// Mitsubishi GX Works2 project: RL8_12-03-62 - LossCode   PLC: Q01U

PROGRAM MAIN  // À¯ÁÊßÈÙ
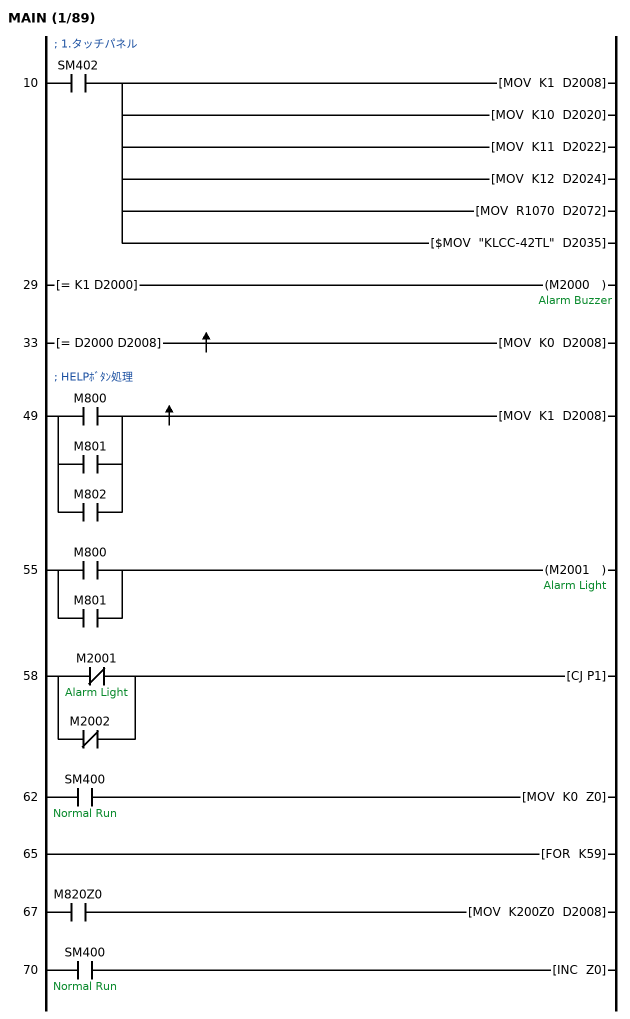
; 1.タッチパネル
; 
10    LD      SM402
      MOV     K1 D2008
      MOV     K10 D2020
      MOV     K11 D2022
      MOV     K12 D2024
      MOV     R1070 D2072
      $MOV    "KLCC-42TL" D2035
29    LD=     K1 D2000
      OUT     M2000  ; Alarm Buzzer
33    LD=     D2000 D2008
      MEP
      MOV     K0 D2008
; HELPﾎﾞﾀﾝ処理
49    LD      M800
      OR      M801
      OR      M802
      MEP
      MOV     K1 D2008
55    LD      M800
      OR      M801
      OUT     M2001  ; Alarm Light
58    LDI     M2001  ; Alarm Light
      ORI     M2002
      CJ      P1
62    LD      SM400  ; Normal Run
      MOV     K0 Z0
65    FOR     K59
67    LD      M820Z0
      MOV     K200Z0 D2008
70    LD      SM400  ; Normal Run
      INC     Z0
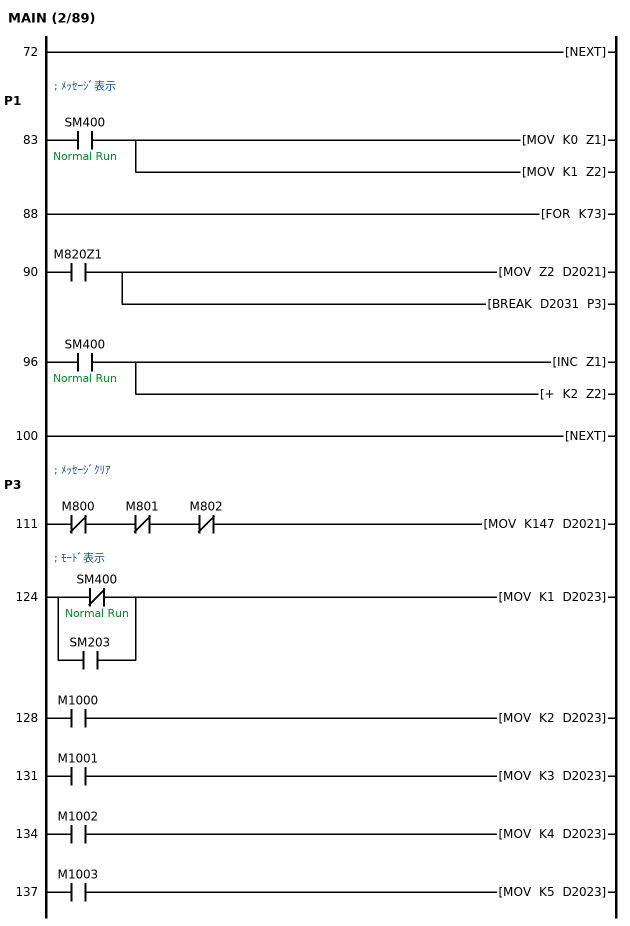
72    NEXT
      P1
; ﾒｯｾｰｼﾞ表示
83    LD      SM400  ; Normal Run
      MOV     K0 Z1
      MOV     K1 Z2
88    FOR     K73
90    LD      M820Z1
      MOV     Z2 D2021
      BREAK   D2031 P3
96    LD      SM400  ; Normal Run
      INC     Z1
      +       K2 Z2
100   NEXT
; ﾒｯｾｰｼﾞｸﾘｱ
      P3
111   LDI     M800
      ANI     M801
      ANI     M802
      MOV     K147 D2021
; ﾓｰﾄﾞ表示
124   LDI     SM400  ; Normal Run
      OR      SM203
      MOV     K1 D2023
128   LD      M1000
      MOV     K2 D2023
131   LD      M1001
      MOV     K3 D2023
134   LD      M1002
      MOV     K4 D2023
137   LD      M1003
      MOV     K5 D2023
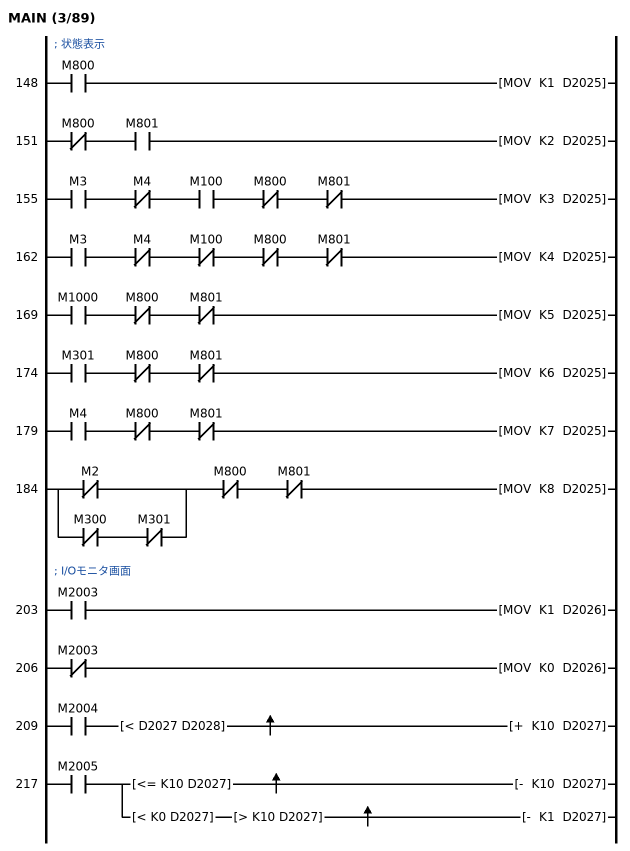
; 状態表示
148   LD      M800
      MOV     K1 D2025
151   LDI     M800
      AND     M801
      MOV     K2 D2025
155   LD      M3
      ANI     M4
      AND     M100
      ANI     M800
      ANI     M801
      MOV     K3 D2025
162   LD      M3
      ANI     M4
      ANI     M100
      ANI     M800
      ANI     M801
      MOV     K4 D2025
169   LD      M1000
      ANI     M800
      ANI     M801
      MOV     K5 D2025
174   LD      M301
      ANI     M800
      ANI     M801
      MOV     K6 D2025
179   LD      M4
      ANI     M800
      ANI     M801
      MOV     K7 D2025
184   LDI     M2
      LDI     M300
      ANI     M301
      ORB
      ANI     M800
      ANI     M801
      MOV     K8 D2025
; I/Oモニタ画面
203   LD      M2003
      MOV     K1 D2026
206   LDI     M2003
      MOV     K0 D2026
209   LD      M2004
      AND<    D2027 D2028
      MEP
      +       K10 D2027
217   LD      M2005
      MPS
      AND<=   K10 D2027
      MEP
      -       K10 D2027
      MPP
      AND<    K0 D2027
      AND>    K10 D2027
      MEP
      -       K1 D2027
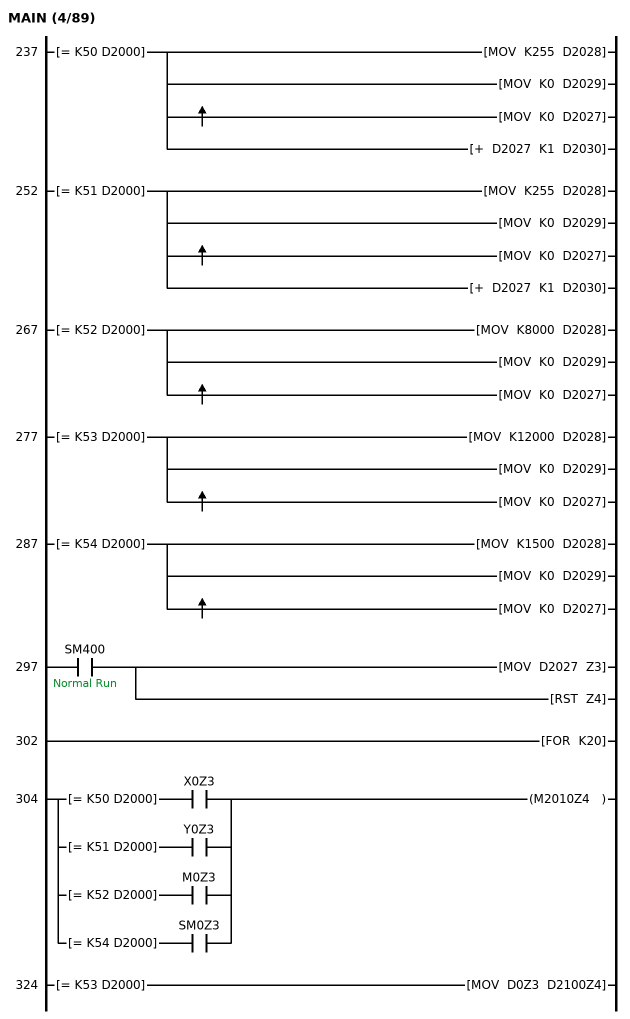
237   LD=     K50 D2000
      MOV     K255 D2028
      MOV     K0 D2029
      MPS
      MEP
      MOV     K0 D2027
      MPP
      +       D2027 K1 D2030
252   LD=     K51 D2000
      MOV     K255 D2028
      MOV     K0 D2029
      MPS
      MEP
      MOV     K0 D2027
      MPP
      +       D2027 K1 D2030
267   LD=     K52 D2000
      MOV     K8000 D2028
      MOV     K0 D2029
      MEP
      MOV     K0 D2027
277   LD=     K53 D2000
      MOV     K12000 D2028
      MOV     K0 D2029
      MEP
      MOV     K0 D2027
287   LD=     K54 D2000
      MOV     K1500 D2028
      MOV     K0 D2029
      MEP
      MOV     K0 D2027
297   LD      SM400  ; Normal Run
      MOV     D2027 Z3
      RST     Z4
302   FOR     K20
304   LD=     K50 D2000
      AND     X0Z3
      LD=     K51 D2000
      AND     Y0Z3
      ORB
      LD=     K52 D2000
      AND     M0Z3
      ORB
      LD=     K54 D2000
      AND     SM0Z3
      ORB
      OUT     M2010Z4
324   LD=     K53 D2000
      MOV     D0Z3 D2100Z4
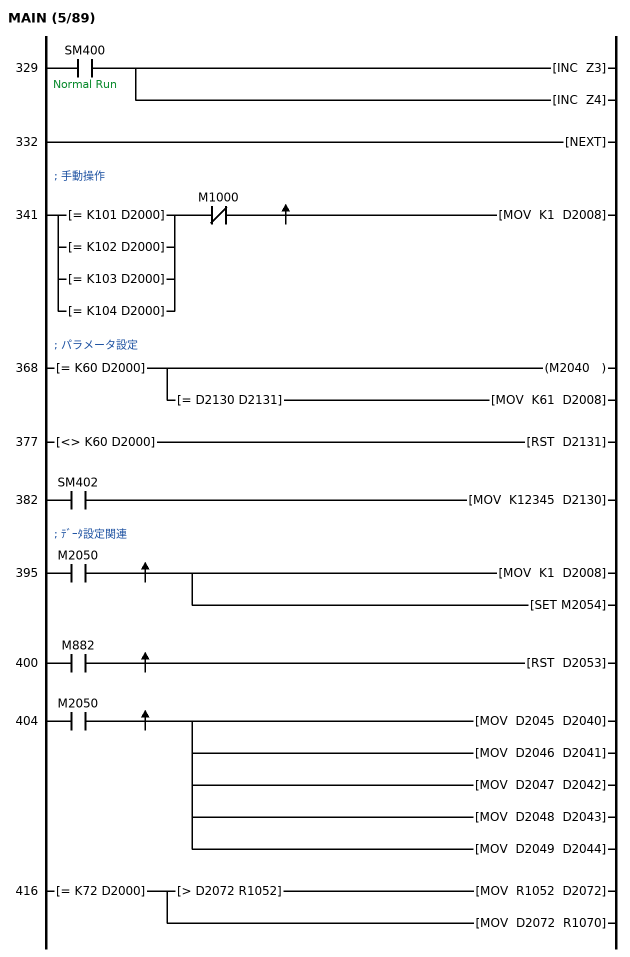
329   LD      SM400  ; Normal Run
      INC     Z3
      INC     Z4
332   NEXT
; 手動操作
341   LD=     K101 D2000
      OR=     K102 D2000
      OR=     K103 D2000
      OR=     K104 D2000
      ANI     M1000
      MEP
      MOV     K1 D2008
; パラメータ設定
368   LD=     K60 D2000
      OUT     M2040
      AND=    D2130 D2131
      MOV     K61 D2008
377   LD<>    K60 D2000
      RST     D2131
382   LD      SM402
      MOV     K12345 D2130
; ﾃﾞｰﾀ設定関連
395   LD      M2050
      MEP
      MOV     K1 D2008
      SET     M2054
400   LD      M882
      MEP
      RST     D2053
404   LD      M2050
      MEP
      MOV     D2045 D2040
      MOV     D2046 D2041
      MOV     D2047 D2042
      MOV     D2048 D2043
      MOV     D2049 D2044
416   LD=     K72 D2000
      MPS
      AND>    D2072 R1052
      MOV     R1052 D2072
      MPP
      MOV     D2072 R1070
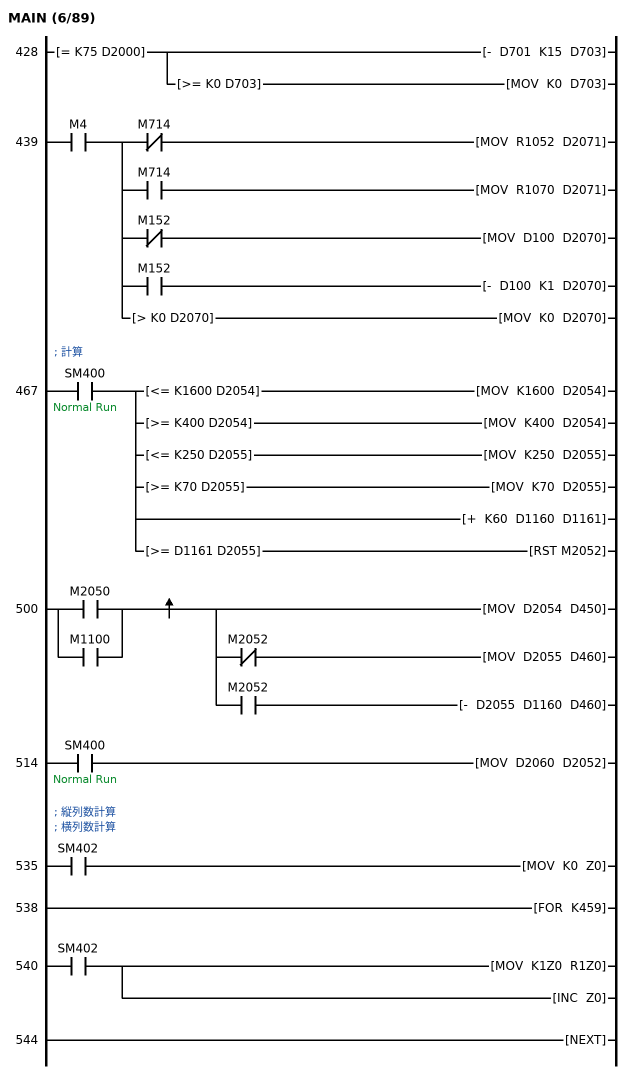
428   LD=     K75 D2000
      -       D701 K15 D703
      AND>=   K0 D703
      MOV     K0 D703
439   LD      M4
      MPS
      ANI     M714
      MOV     R1052 D2071
      MRD
      AND     M714
      MOV     R1070 D2071
      MRD
      ANI     M152
      MOV     D100 D2070
      MRD
      AND     M152
      -       D100 K1 D2070
      MPP
      AND>    K0 D2070
      MOV     K0 D2070
; 計算
467   LD      SM400  ; Normal Run
      MPS
      AND<=   K1600 D2054
      MOV     K1600 D2054
      MRD
      AND>=   K400 D2054
      MOV     K400 D2054
      MRD
      AND<=   K250 D2055
      MOV     K250 D2055
      MRD
      AND>=   K70 D2055
      MOV     K70 D2055
      MPP
      +       K60 D1160 D1161
      AND>=   D1161 D2055
      RST     M2052
500   LD      M2050
      OR      M1100
      MEP
      MOV     D2054 D450
      MPS
      ANI     M2052
      MOV     D2055 D460
      MPP
      AND     M2052
      -       D2055 D1160 D460
514   LD      SM400  ; Normal Run
      MOV     D2060 D2052
; 縦列数計算
; 横列数計算
535   LD      SM402
      MOV     K0 Z0
538   FOR     K459
540   LD      SM402
      MOV     K1Z0 R1Z0
      INC     Z0
544   NEXT
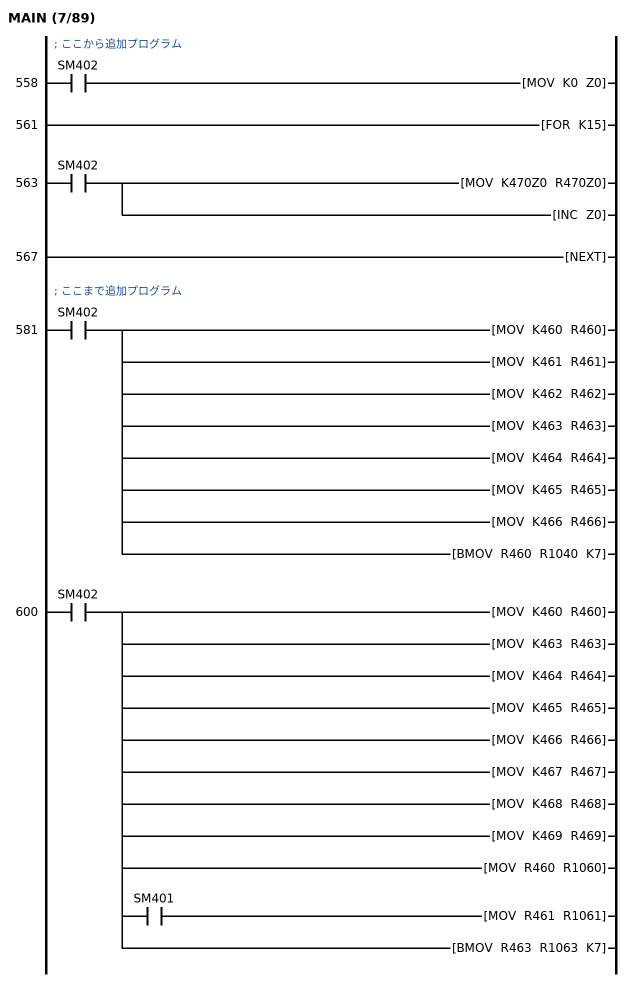
; ここから追加プログラム
558   LD      SM402
      MOV     K0 Z0
561   FOR     K15
563   LD      SM402
      MOV     K470Z0 R470Z0
      INC     Z0
567   NEXT
; ここまで追加プログラム
581   LD      SM402
      MOV     K460 R460
      MOV     K461 R461
      MOV     K462 R462
      MOV     K463 R463
      MOV     K464 R464
      MOV     K465 R465
      MOV     K466 R466
      BMOV    R460 R1040 K7
600   LD      SM402
      MOV     K460 R460
      MOV     K463 R463
      MOV     K464 R464
      MOV     K465 R465
      MOV     K466 R466
      MOV     K467 R467
      MOV     K468 R468
      MOV     K469 R469
      MOV     R460 R1060
      MPS
      AND     SM401
      MOV     R461 R1061
      MPP
      BMOV    R463 R1063 K7
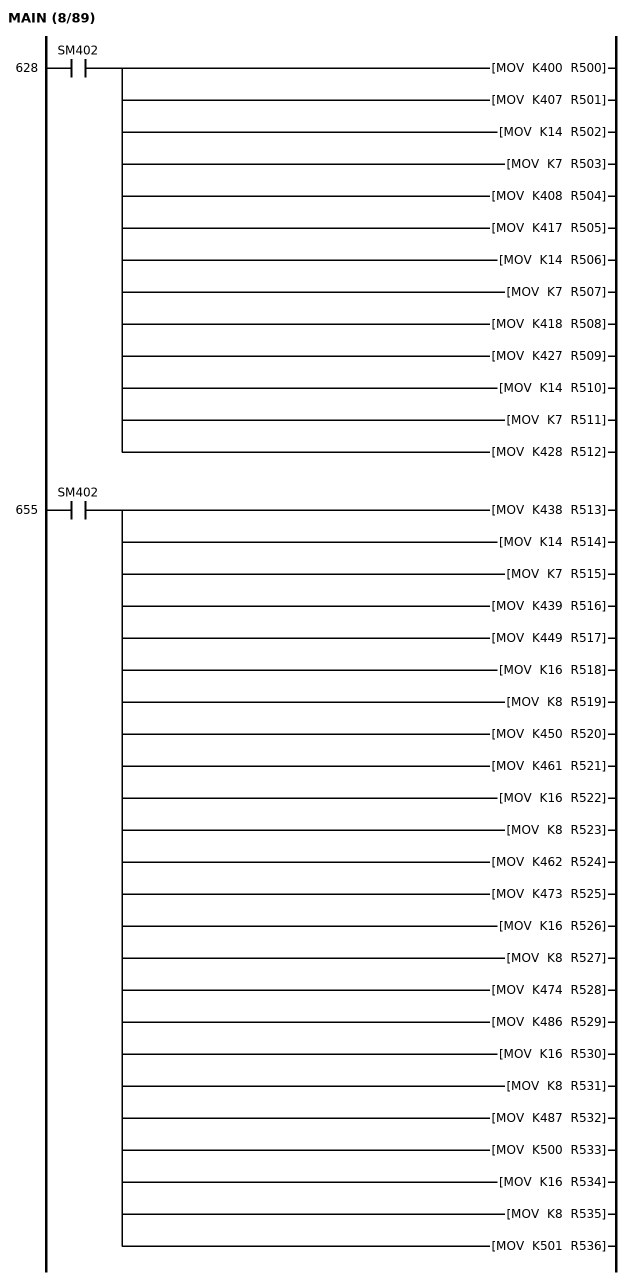
628   LD      SM402
      MOV     K400 R500
      MOV     K407 R501
      MOV     K14 R502
      MOV     K7 R503
      MOV     K408 R504
      MOV     K417 R505
      MOV     K14 R506
      MOV     K7 R507
      MOV     K418 R508
      MOV     K427 R509
      MOV     K14 R510
      MOV     K7 R511
      MOV     K428 R512
655   LD      SM402
      MOV     K438 R513
      MOV     K14 R514
      MOV     K7 R515
      MOV     K439 R516
      MOV     K449 R517
      MOV     K16 R518
      MOV     K8 R519
      MOV     K450 R520
      MOV     K461 R521
      MOV     K16 R522
      MOV     K8 R523
      MOV     K462 R524
      MOV     K473 R525
      MOV     K16 R526
      MOV     K8 R527
      MOV     K474 R528
      MOV     K486 R529
      MOV     K16 R530
      MOV     K8 R531
      MOV     K487 R532
      MOV     K500 R533
      MOV     K16 R534
      MOV     K8 R535
      MOV     K501 R536
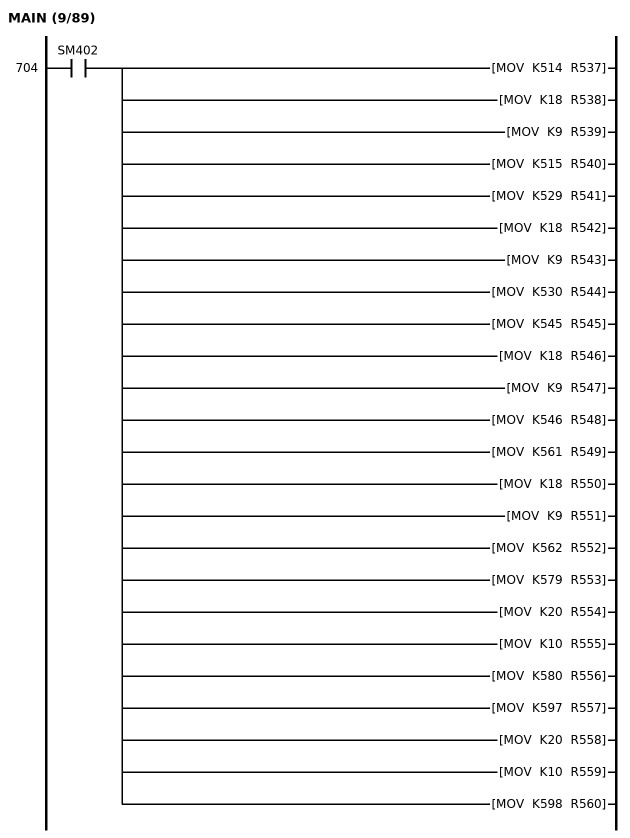
704   LD      SM402
      MOV     K514 R537
      MOV     K18 R538
      MOV     K9 R539
      MOV     K515 R540
      MOV     K529 R541
      MOV     K18 R542
      MOV     K9 R543
      MOV     K530 R544
      MOV     K545 R545
      MOV     K18 R546
      MOV     K9 R547
      MOV     K546 R548
      MOV     K561 R549
      MOV     K18 R550
      MOV     K9 R551
      MOV     K562 R552
      MOV     K579 R553
      MOV     K20 R554
      MOV     K10 R555
      MOV     K580 R556
      MOV     K597 R557
      MOV     K20 R558
      MOV     K10 R559
      MOV     K598 R560
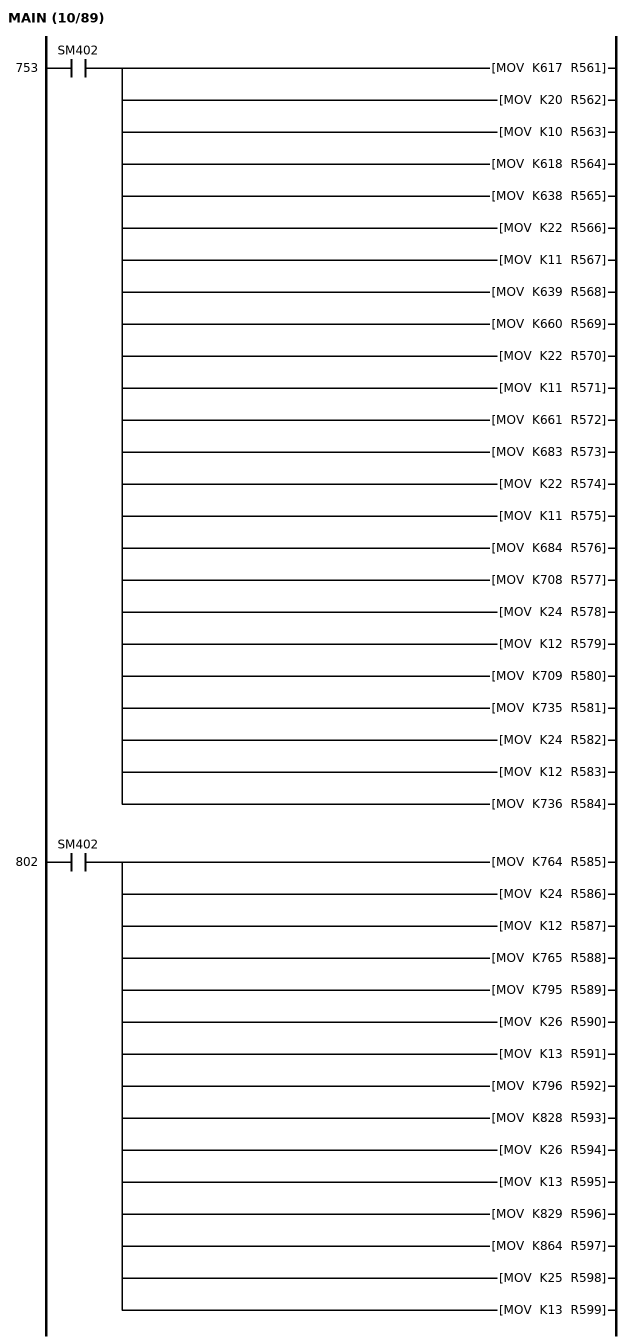
753   LD      SM402
      MOV     K617 R561
      MOV     K20 R562
      MOV     K10 R563
      MOV     K618 R564
      MOV     K638 R565
      MOV     K22 R566
      MOV     K11 R567
      MOV     K639 R568
      MOV     K660 R569
      MOV     K22 R570
      MOV     K11 R571
      MOV     K661 R572
      MOV     K683 R573
      MOV     K22 R574
      MOV     K11 R575
      MOV     K684 R576
      MOV     K708 R577
      MOV     K24 R578
      MOV     K12 R579
      MOV     K709 R580
      MOV     K735 R581
      MOV     K24 R582
      MOV     K12 R583
      MOV     K736 R584
802   LD      SM402
      MOV     K764 R585
      MOV     K24 R586
      MOV     K12 R587
      MOV     K765 R588
      MOV     K795 R589
      MOV     K26 R590
      MOV     K13 R591
      MOV     K796 R592
      MOV     K828 R593
      MOV     K26 R594
      MOV     K13 R595
      MOV     K829 R596
      MOV     K864 R597
      MOV     K25 R598
      MOV     K13 R599
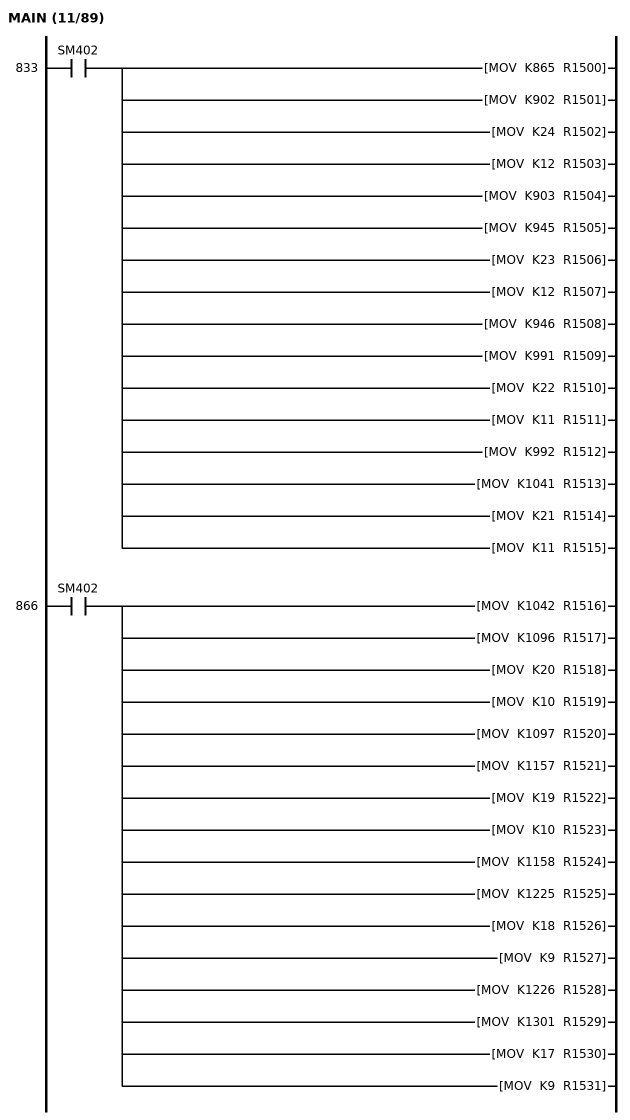
833   LD      SM402
      MOV     K865 R1500
      MOV     K902 R1501
      MOV     K24 R1502
      MOV     K12 R1503
      MOV     K903 R1504
      MOV     K945 R1505
      MOV     K23 R1506
      MOV     K12 R1507
      MOV     K946 R1508
      MOV     K991 R1509
      MOV     K22 R1510
      MOV     K11 R1511
      MOV     K992 R1512
      MOV     K1041 R1513
      MOV     K21 R1514
      MOV     K11 R1515
866   LD      SM402
      MOV     K1042 R1516
      MOV     K1096 R1517
      MOV     K20 R1518
      MOV     K10 R1519
      MOV     K1097 R1520
      MOV     K1157 R1521
      MOV     K19 R1522
      MOV     K10 R1523
      MOV     K1158 R1524
      MOV     K1225 R1525
      MOV     K18 R1526
      MOV     K9 R1527
      MOV     K1226 R1528
      MOV     K1301 R1529
      MOV     K17 R1530
      MOV     K9 R1531
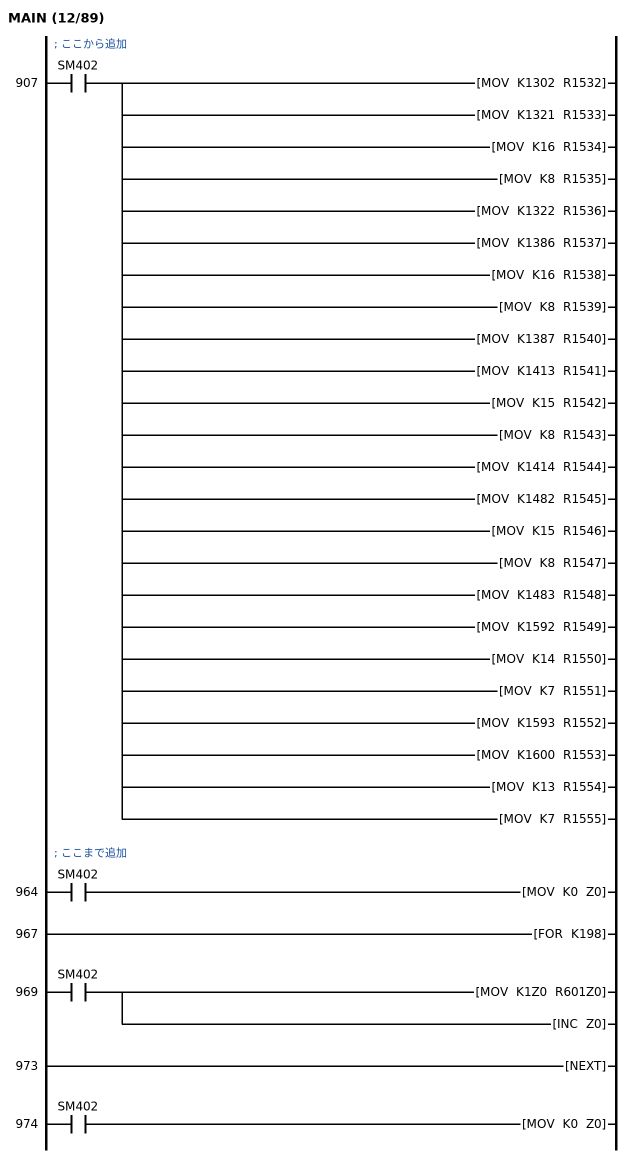
; ここから追加
907   LD      SM402
      MOV     K1302 R1532
      MOV     K1321 R1533
      MOV     K16 R1534
      MOV     K8 R1535
      MOV     K1322 R1536
      MOV     K1386 R1537
      MOV     K16 R1538
      MOV     K8 R1539
      MOV     K1387 R1540
      MOV     K1413 R1541
      MOV     K15 R1542
      MOV     K8 R1543
      MOV     K1414 R1544
      MOV     K1482 R1545
      MOV     K15 R1546
      MOV     K8 R1547
      MOV     K1483 R1548
      MOV     K1592 R1549
      MOV     K14 R1550
      MOV     K7 R1551
      MOV     K1593 R1552
      MOV     K1600 R1553
      MOV     K13 R1554
      MOV     K7 R1555
; ここまで追加
964   LD      SM402
      MOV     K0 Z0
967   FOR     K198
969   LD      SM402
      MOV     K1Z0 R601Z0
      INC     Z0
973   NEXT
974   LD      SM402
      MOV     K0 Z0
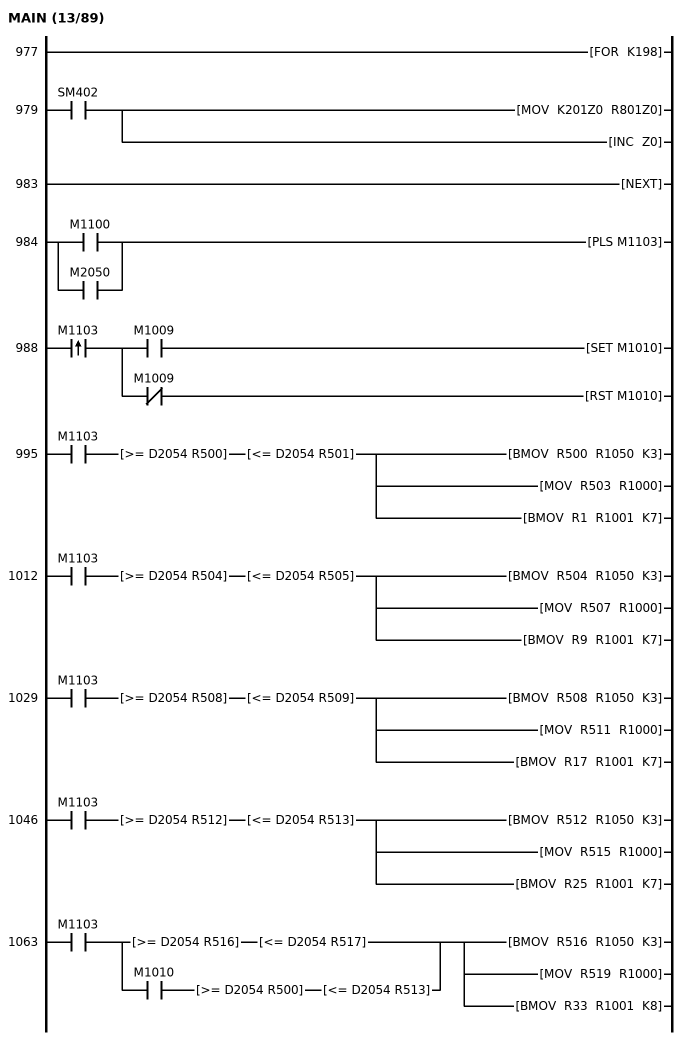
977   FOR     K198
979   LD      SM402
      MOV     K201Z0 R801Z0
      INC     Z0
983   NEXT
984   LD      M1100
      OR      M2050
      PLS     M1103
988   LDP     M1103
      MPS
      AND     M1009
      SET     M1010
      MPP
      ANI     M1009
      RST     M1010
995   LD      M1103
      AND>=   D2054 R500
      AND<=   D2054 R501
      BMOV    R500 R1050 K3
      MOV     R503 R1000
      BMOV    R1 R1001 K7
1012  LD      M1103
      AND>=   D2054 R504
      AND<=   D2054 R505
      BMOV    R504 R1050 K3
      MOV     R507 R1000
      BMOV    R9 R1001 K7
1029  LD      M1103
      AND>=   D2054 R508
      AND<=   D2054 R509
      BMOV    R508 R1050 K3
      MOV     R511 R1000
      BMOV    R17 R1001 K7
1046  LD      M1103
      AND>=   D2054 R512
      AND<=   D2054 R513
      BMOV    R512 R1050 K3
      MOV     R515 R1000
      BMOV    R25 R1001 K7
1063  LD      M1103
      LD>=    D2054 R516
      AND<=   D2054 R517
      LD      M1010
      AND>=   D2054 R500
      AND<=   D2054 R513
      ORB
      ANB
      BMOV    R516 R1050 K3
      MOV     R519 R1000
      BMOV    R33 R1001 K8
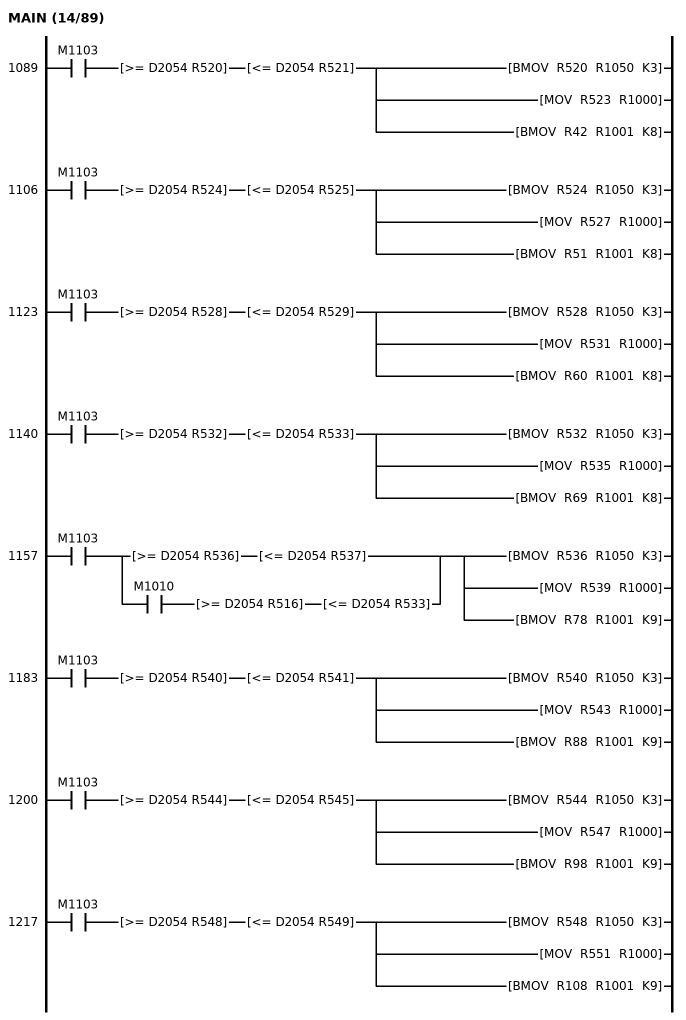
1089  LD      M1103
      AND>=   D2054 R520
      AND<=   D2054 R521
      BMOV    R520 R1050 K3
      MOV     R523 R1000
      BMOV    R42 R1001 K8
1106  LD      M1103
      AND>=   D2054 R524
      AND<=   D2054 R525
      BMOV    R524 R1050 K3
      MOV     R527 R1000
      BMOV    R51 R1001 K8
1123  LD      M1103
      AND>=   D2054 R528
      AND<=   D2054 R529
      BMOV    R528 R1050 K3
      MOV     R531 R1000
      BMOV    R60 R1001 K8
1140  LD      M1103
      AND>=   D2054 R532
      AND<=   D2054 R533
      BMOV    R532 R1050 K3
      MOV     R535 R1000
      BMOV    R69 R1001 K8
1157  LD      M1103
      LD>=    D2054 R536
      AND<=   D2054 R537
      LD      M1010
      AND>=   D2054 R516
      AND<=   D2054 R533
      ORB
      ANB
      BMOV    R536 R1050 K3
      MOV     R539 R1000
      BMOV    R78 R1001 K9
1183  LD      M1103
      AND>=   D2054 R540
      AND<=   D2054 R541
      BMOV    R540 R1050 K3
      MOV     R543 R1000
      BMOV    R88 R1001 K9
1200  LD      M1103
      AND>=   D2054 R544
      AND<=   D2054 R545
      BMOV    R544 R1050 K3
      MOV     R547 R1000
      BMOV    R98 R1001 K9
1217  LD      M1103
      AND>=   D2054 R548
      AND<=   D2054 R549
      BMOV    R548 R1050 K3
      MOV     R551 R1000
      BMOV    R108 R1001 K9
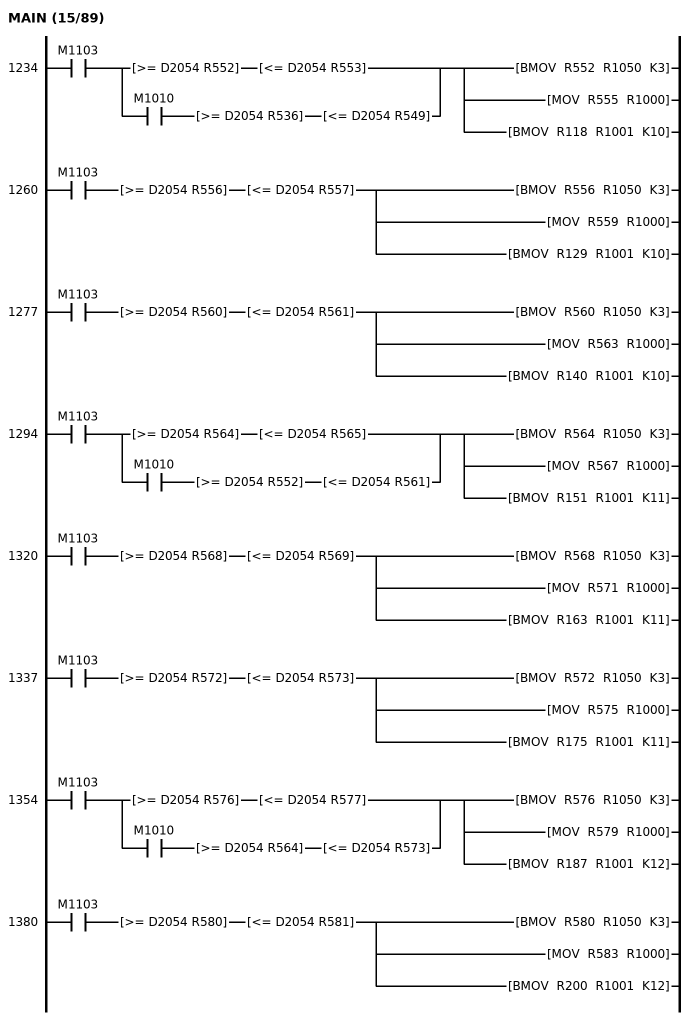
1234  LD      M1103
      LD>=    D2054 R552
      AND<=   D2054 R553
      LD      M1010
      AND>=   D2054 R536
      AND<=   D2054 R549
      ORB
      ANB
      BMOV    R552 R1050 K3
      MOV     R555 R1000
      BMOV    R118 R1001 K10
1260  LD      M1103
      AND>=   D2054 R556
      AND<=   D2054 R557
      BMOV    R556 R1050 K3
      MOV     R559 R1000
      BMOV    R129 R1001 K10
1277  LD      M1103
      AND>=   D2054 R560
      AND<=   D2054 R561
      BMOV    R560 R1050 K3
      MOV     R563 R1000
      BMOV    R140 R1001 K10
1294  LD      M1103
      LD>=    D2054 R564
      AND<=   D2054 R565
      LD      M1010
      AND>=   D2054 R552
      AND<=   D2054 R561
      ORB
      ANB
      BMOV    R564 R1050 K3
      MOV     R567 R1000
      BMOV    R151 R1001 K11
1320  LD      M1103
      AND>=   D2054 R568
      AND<=   D2054 R569
      BMOV    R568 R1050 K3
      MOV     R571 R1000
      BMOV    R163 R1001 K11
1337  LD      M1103
      AND>=   D2054 R572
      AND<=   D2054 R573
      BMOV    R572 R1050 K3
      MOV     R575 R1000
      BMOV    R175 R1001 K11
1354  LD      M1103
      LD>=    D2054 R576
      AND<=   D2054 R577
      LD      M1010
      AND>=   D2054 R564
      AND<=   D2054 R573
      ORB
      ANB
      BMOV    R576 R1050 K3
      MOV     R579 R1000
      BMOV    R187 R1001 K12
1380  LD      M1103
      AND>=   D2054 R580
      AND<=   D2054 R581
      BMOV    R580 R1050 K3
      MOV     R583 R1000
      BMOV    R200 R1001 K12
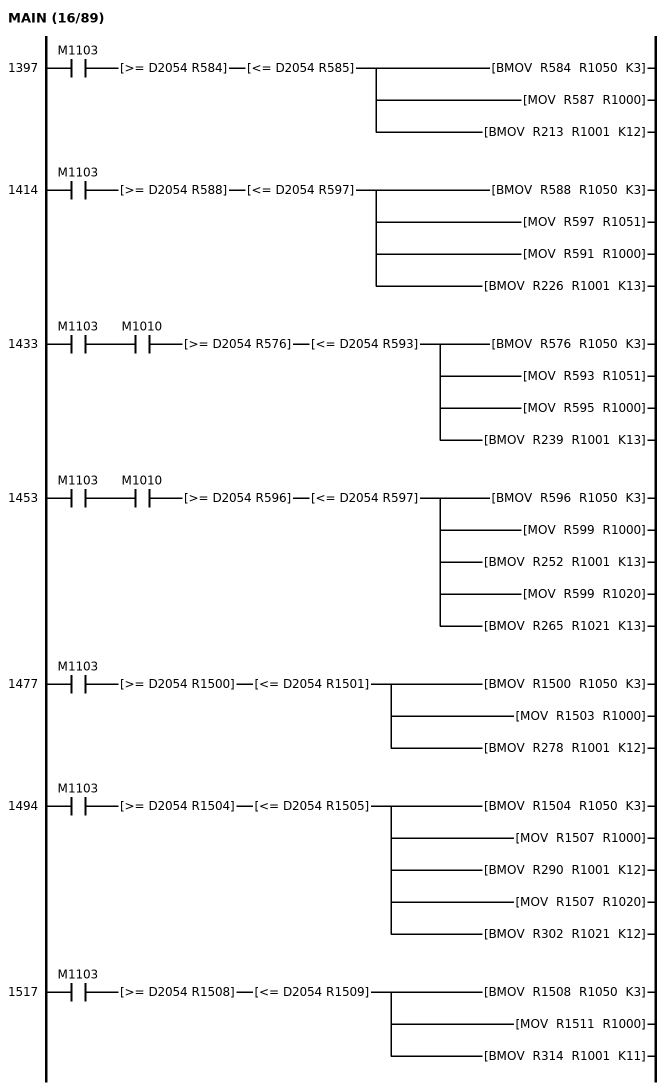
1397  LD      M1103
      AND>=   D2054 R584
      AND<=   D2054 R585
      BMOV    R584 R1050 K3
      MOV     R587 R1000
      BMOV    R213 R1001 K12
1414  LD      M1103
      AND>=   D2054 R588
      AND<=   D2054 R597
      BMOV    R588 R1050 K3
      MOV     R597 R1051
      MOV     R591 R1000
      BMOV    R226 R1001 K13
1433  LD      M1103
      AND     M1010
      AND>=   D2054 R576
      AND<=   D2054 R593
      BMOV    R576 R1050 K3
      MOV     R593 R1051
      MOV     R595 R1000
      BMOV    R239 R1001 K13
1453  LD      M1103
      AND     M1010
      AND>=   D2054 R596
      AND<=   D2054 R597
      BMOV    R596 R1050 K3
      MOV     R599 R1000
      BMOV    R252 R1001 K13
      MOV     R599 R1020
      BMOV    R265 R1021 K13
1477  LD      M1103
      AND>=   D2054 R1500
      AND<=   D2054 R1501
      BMOV    R1500 R1050 K3
      MOV     R1503 R1000
      BMOV    R278 R1001 K12
1494  LD      M1103
      AND>=   D2054 R1504
      AND<=   D2054 R1505
      BMOV    R1504 R1050 K3
      MOV     R1507 R1000
      BMOV    R290 R1001 K12
      MOV     R1507 R1020
      BMOV    R302 R1021 K12
1517  LD      M1103
      AND>=   D2054 R1508
      AND<=   D2054 R1509
      BMOV    R1508 R1050 K3
      MOV     R1511 R1000
      BMOV    R314 R1001 K11
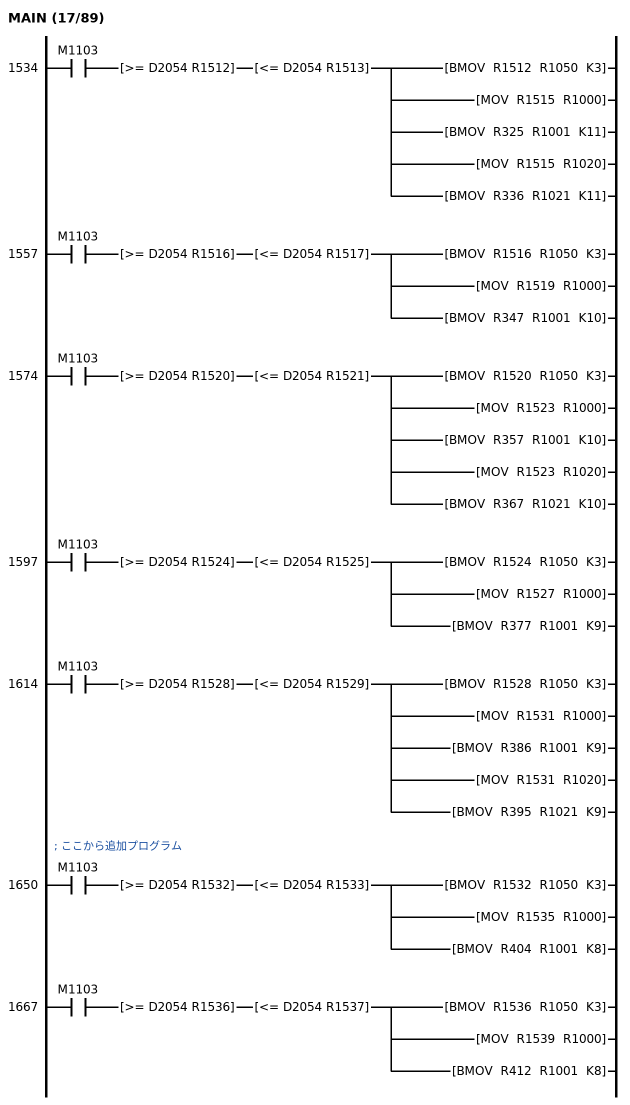
1534  LD      M1103
      AND>=   D2054 R1512
      AND<=   D2054 R1513
      BMOV    R1512 R1050 K3
      MOV     R1515 R1000
      BMOV    R325 R1001 K11
      MOV     R1515 R1020
      BMOV    R336 R1021 K11
1557  LD      M1103
      AND>=   D2054 R1516
      AND<=   D2054 R1517
      BMOV    R1516 R1050 K3
      MOV     R1519 R1000
      BMOV    R347 R1001 K10
1574  LD      M1103
      AND>=   D2054 R1520
      AND<=   D2054 R1521
      BMOV    R1520 R1050 K3
      MOV     R1523 R1000
      BMOV    R357 R1001 K10
      MOV     R1523 R1020
      BMOV    R367 R1021 K10
1597  LD      M1103
      AND>=   D2054 R1524
      AND<=   D2054 R1525
      BMOV    R1524 R1050 K3
      MOV     R1527 R1000
      BMOV    R377 R1001 K9
1614  LD      M1103
      AND>=   D2054 R1528
      AND<=   D2054 R1529
      BMOV    R1528 R1050 K3
      MOV     R1531 R1000
      BMOV    R386 R1001 K9
      MOV     R1531 R1020
      BMOV    R395 R1021 K9
; ここから追加プログラム
1650  LD      M1103
      AND>=   D2054 R1532
      AND<=   D2054 R1533
      BMOV    R1532 R1050 K3
      MOV     R1535 R1000
      BMOV    R404 R1001 K8
1667  LD      M1103
      AND>=   D2054 R1536
      AND<=   D2054 R1537
      BMOV    R1536 R1050 K3
      MOV     R1539 R1000
      BMOV    R412 R1001 K8
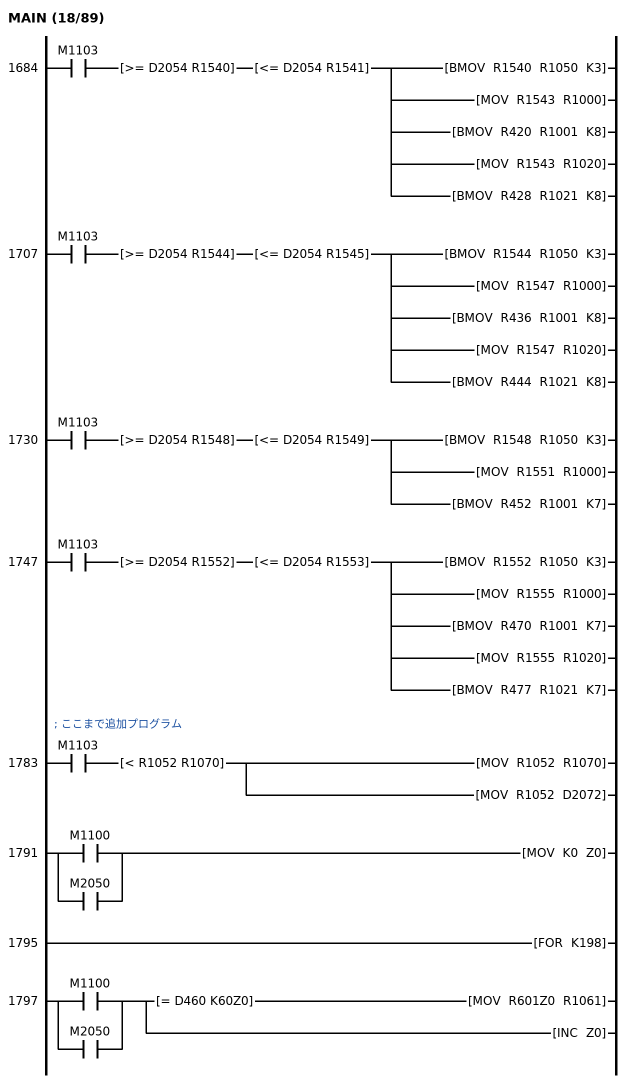
1684  LD      M1103
      AND>=   D2054 R1540
      AND<=   D2054 R1541
      BMOV    R1540 R1050 K3
      MOV     R1543 R1000
      BMOV    R420 R1001 K8
      MOV     R1543 R1020
      BMOV    R428 R1021 K8
1707  LD      M1103
      AND>=   D2054 R1544
      AND<=   D2054 R1545
      BMOV    R1544 R1050 K3
      MOV     R1547 R1000
      BMOV    R436 R1001 K8
      MOV     R1547 R1020
      BMOV    R444 R1021 K8
1730  LD      M1103
      AND>=   D2054 R1548
      AND<=   D2054 R1549
      BMOV    R1548 R1050 K3
      MOV     R1551 R1000
      BMOV    R452 R1001 K7
1747  LD      M1103
      AND>=   D2054 R1552
      AND<=   D2054 R1553
      BMOV    R1552 R1050 K3
      MOV     R1555 R1000
      BMOV    R470 R1001 K7
      MOV     R1555 R1020
      BMOV    R477 R1021 K7
; ここまで追加プログラム
1783  LD      M1103
      AND<    R1052 R1070
      MOV     R1052 R1070
      MOV     R1052 D2072
1791  LD      M1100
      OR      M2050
      MOV     K0 Z0
1795  FOR     K198
1797  LD      M1100
      OR      M2050
      MPS
      AND=    D460 K60Z0
      MOV     R601Z0 R1061
      MPP
      INC     Z0
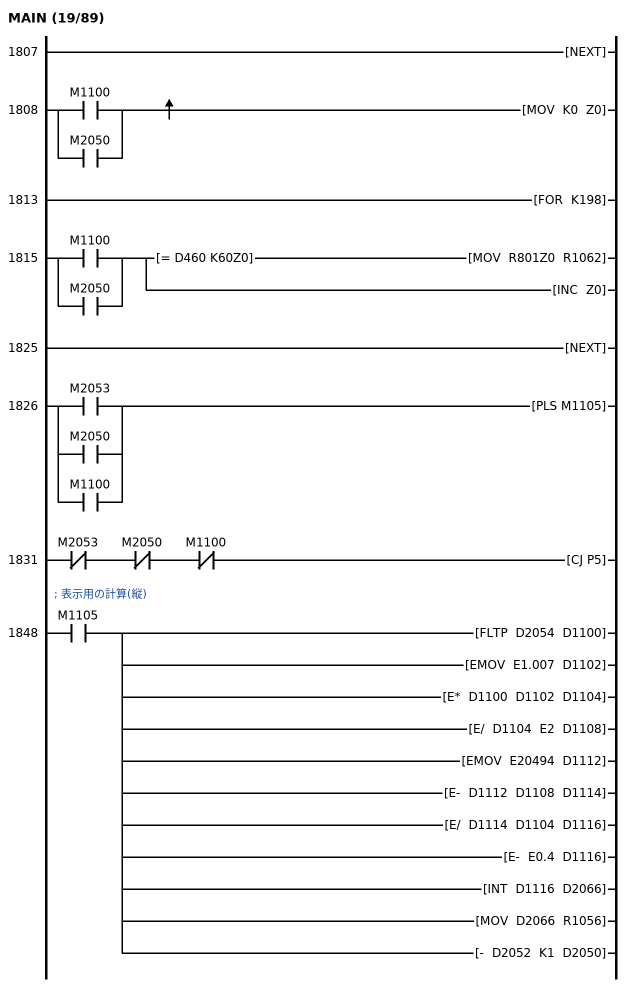
1807  NEXT
1808  LD      M1100
      OR      M2050
      MEP
      MOV     K0 Z0
1813  FOR     K198
1815  LD      M1100
      OR      M2050
      MPS
      AND=    D460 K60Z0
      MOV     R801Z0 R1062
      MPP
      INC     Z0
1825  NEXT
1826  LD      M2053
      OR      M2050
      OR      M1100
      PLS     M1105
1831  LDI     M2053
      ANI     M2050
      ANI     M1100
      CJ      P5
; 表示用の計算(縦)
1848  LD      M1105
      FLTP    D2054 D1100
      EMOV    E1.007 D1102
      E*      D1100 D1102 D1104
      E/      D1104 E2 D1108
      EMOV    E20494 D1112
      E-      D1112 D1108 D1114
      E/      D1114 D1104 D1116
      E-      E0.4 D1116
      INT     D1116 D2066
      MOV     D2066 R1056
      -       D2052 K1 D2050
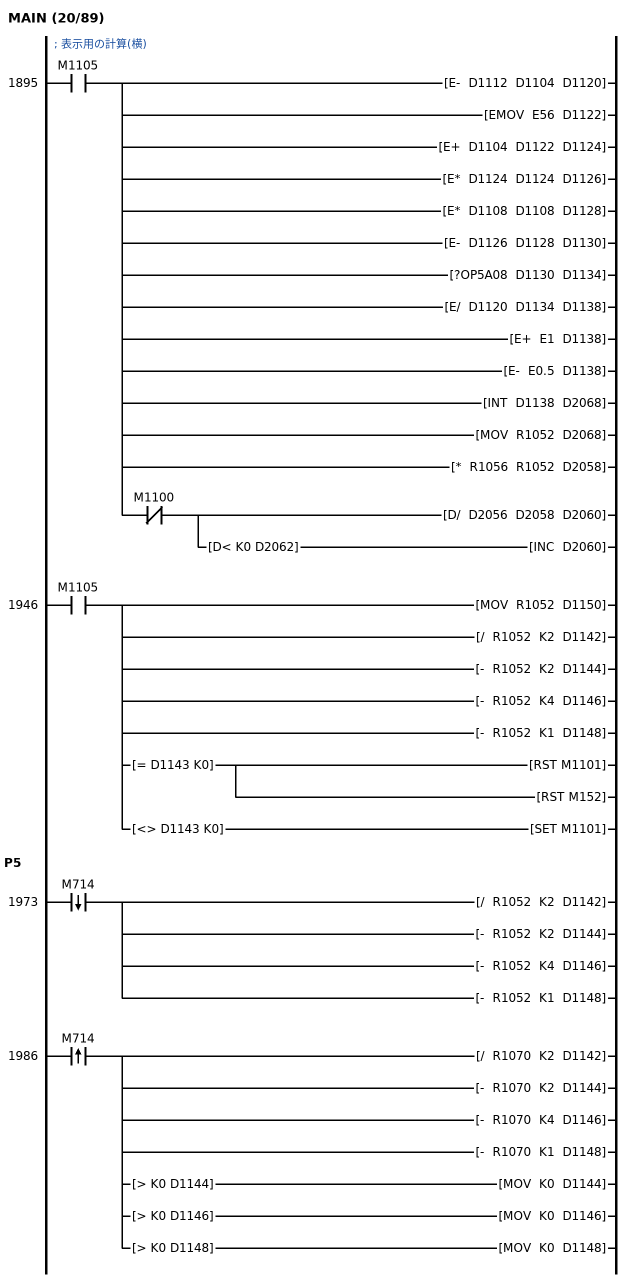
; 表示用の計算(横)
1895  LD      M1105
      E-      D1112 D1104 D1120
      EMOV    E56 D1122
      E+      D1104 D1122 D1124
      E*      D1124 D1124 D1126
      E*      D1108 D1108 D1128
      E-      D1126 D1128 D1130
      ?OP5A08 D1130 D1134
      E/      D1120 D1134 D1138
      E+      E1 D1138
      E-      E0.5 D1138
      INT     D1138 D2068
      MOV     R1052 D2068
      *       R1056 R1052 D2058
      ANI     M1100
      D/      D2056 D2058 D2060
      ANDD<   K0 D2062
      INC     D2060
1946  LD      M1105
      MOV     R1052 D1150
      /       R1052 K2 D1142
      -       R1052 K2 D1144
      -       R1052 K4 D1146
      -       R1052 K1 D1148
      MPS
      AND=    D1143 K0
      RST     M1101
      RST     M152
      MPP
      AND<>   D1143 K0
      SET     M1101
      P5
1973  LDF     M714
      /       R1052 K2 D1142
      -       R1052 K2 D1144
      -       R1052 K4 D1146
      -       R1052 K1 D1148
1986  LDP     M714
      /       R1070 K2 D1142
      -       R1070 K2 D1144
      -       R1070 K4 D1146
      -       R1070 K1 D1148
      MPS
      AND>    K0 D1144
      MOV     K0 D1144
      MRD
      AND>    K0 D1146
      MOV     K0 D1146
      MPP
      AND>    K0 D1148
      MOV     K0 D1148
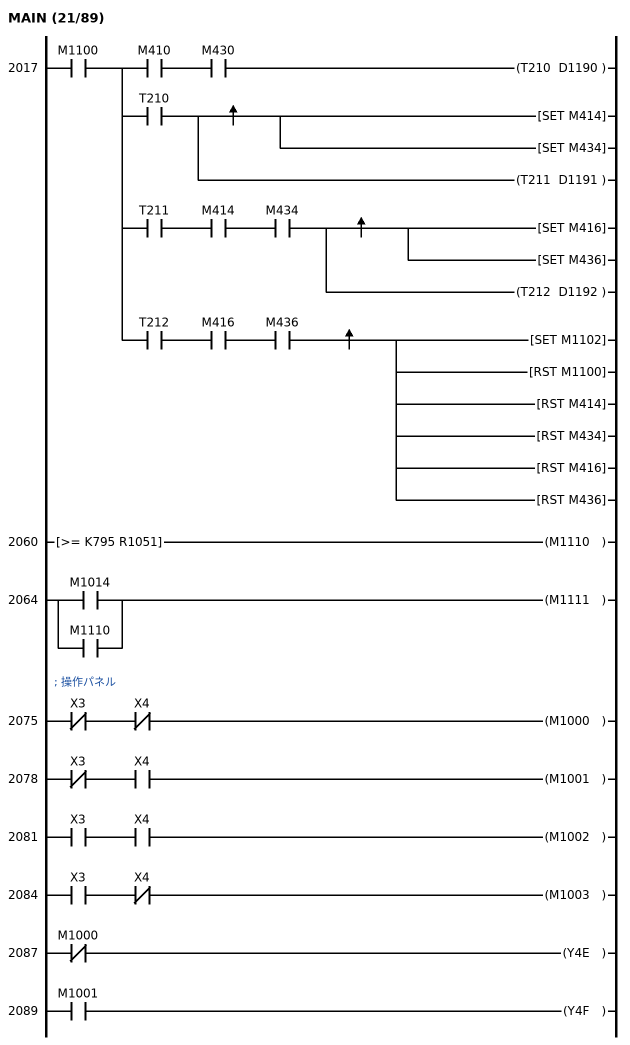
2017  LD      M1100
      MPS
      AND     M410
      AND     M430
      OUT     T210 D1190
      MRD
      AND     T210
      MPS
      MEP
      SET     M414
      SET     M434
      MPP
      OUT     T211 D1191
      MRD
      AND     T211
      AND     M414
      AND     M434
      MPS
      MEP
      SET     M416
      SET     M436
      MPP
      OUT     T212 D1192
      MPP
      AND     T212
      AND     M416
      AND     M436
      MEP
      SET     M1102
      RST     M1100
      RST     M414
      RST     M434
      RST     M416
      RST     M436
2060  LD>=    K795 R1051
      OUT     M1110
2064  LD      M1014
      OR      M1110
      OUT     M1111
; 操作パネル
; 
2075  LDI     X3
      ANI     X4
      OUT     M1000
2078  LDI     X3
      AND     X4
      OUT     M1001
2081  LD      X3
      AND     X4
      OUT     M1002
2084  LD      X3
      ANI     X4
      OUT     M1003
2087  LDI     M1000
      OUT     Y4E
2089  LD      M1001
      OUT     Y4F
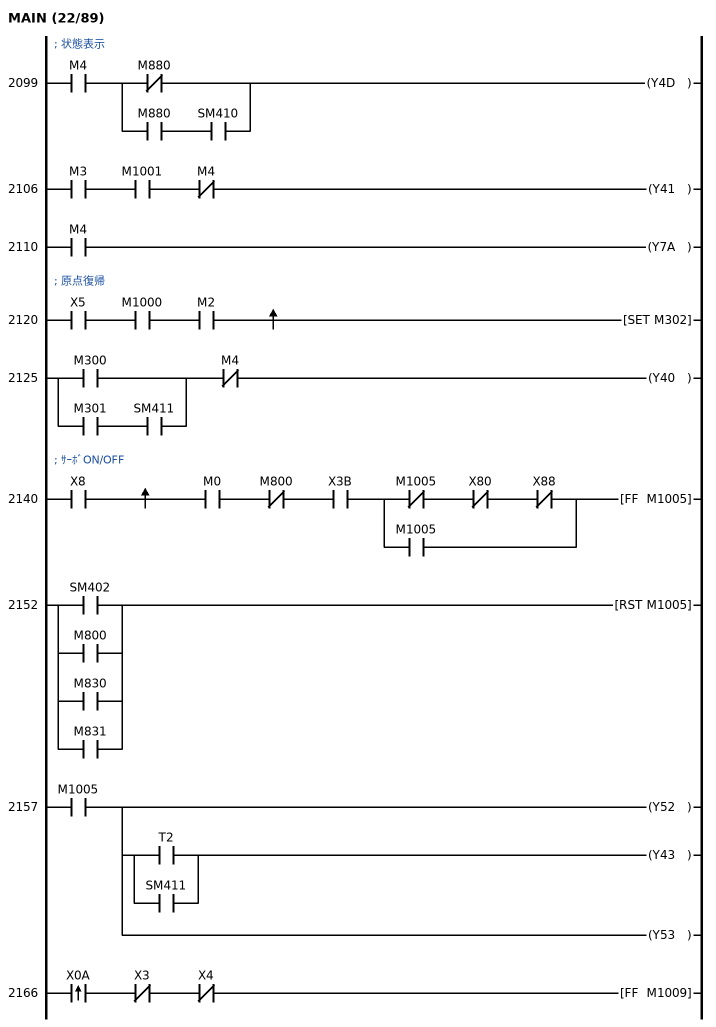
; 状態表示
2099  LD      M4
      LDI     M880
      LD      M880
      AND     SM410
      ORB
      ANB
      OUT     Y4D
2106  LD      M3
      AND     M1001
      ANI     M4
      OUT     Y41
2110  LD      M4
      OUT     Y7A
; 原点復帰
2120  LD      X5
      AND     M1000
      AND     M2
      MEP
      SET     M302
2125  LD      M300
      LD      M301
      AND     SM411
      ORB
      ANI     M4
      OUT     Y40
; ｻｰﾎﾞON/OFF
2140  LD      X8
      MEP
      AND     M0
      ANI     M800
      AND     X3B
      LDI     M1005
      ANI     X80
      ANI     X88
      OR      M1005
      ANB
      FF      M1005
2152  LD      SM402
      OR      M800
      OR      M830
      OR      M831
      RST     M1005
2157  LD      M1005
      OUT     Y52
      MPS
      LD      T2
      OR      SM411
      ANB
      OUT     Y43
      MPP
      OUT     Y53
2166  LDP     X0A
      ANI     X3
      ANI     X4
      FF      M1009
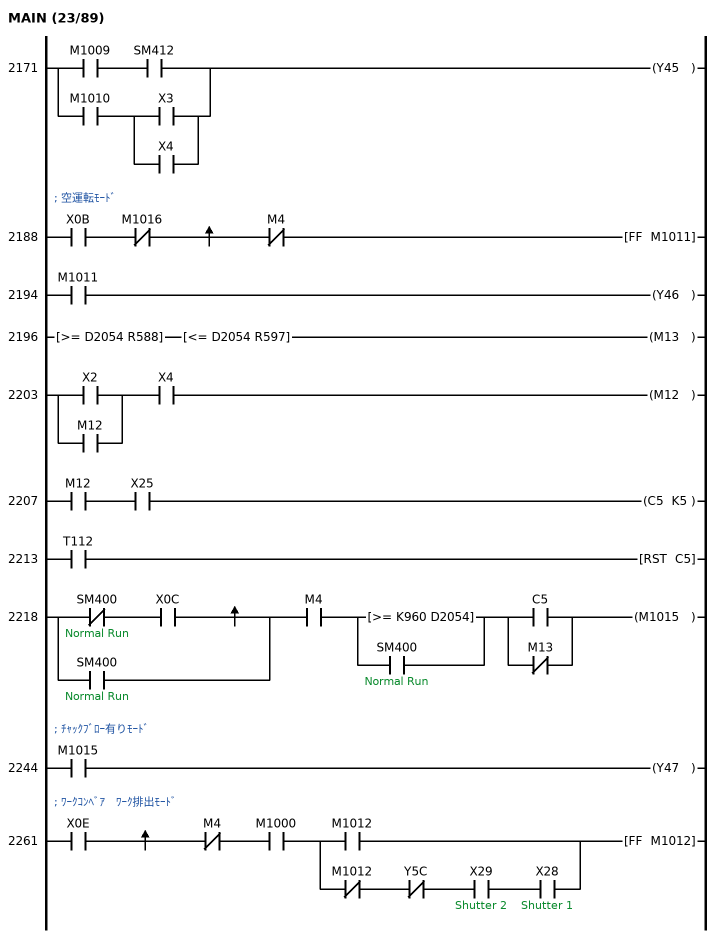
2171  LD      M1009
      AND     SM412
      LD      M1010
      LD      X3
      OR      X4
      ANB
      ORB
      OUT     Y45
; 空運転ﾓｰﾄﾞ
2188  LD      X0B
      ANI     M1016
      MEP
      ANI     M4
      FF      M1011
2194  LD      M1011
      OUT     Y46
2196  LD>=    D2054 R588
      AND<=   D2054 R597
      OUT     M13
2203  LD      X2
      OR      M12
      AND     X4
      OUT     M12
2207  LD      M12
      AND     X25
      OUT     C5 K5
2213  LD      T112
      RST     C5
2218  LDI     SM400  ; Normal Run
      AND     X0C
      MEP
      OR      SM400  ; Normal Run
      AND     M4
      LD>=    K960 D2054
      OR      SM400  ; Normal Run
      ANB
      LD      C5
      ORI     M13
      ANB
      OUT     M1015
; ﾁｬｯｸﾌﾞﾛｰ有りﾓｰﾄﾞ
2244  LD      M1015
      OUT     Y47
; ﾜｰｸｺﾝﾍﾞｱ　ﾜｰｸ排出ﾓｰﾄﾞ
2261  LD      X0E
      MEP
      ANI     M4
      AND     M1000
      LD      M1012
      LDI     M1012
      ANI     Y5C
      AND     X29  ; Shutter 2
      AND     X28  ; Shutter 1
      ORB
      ANB
      FF      M1012
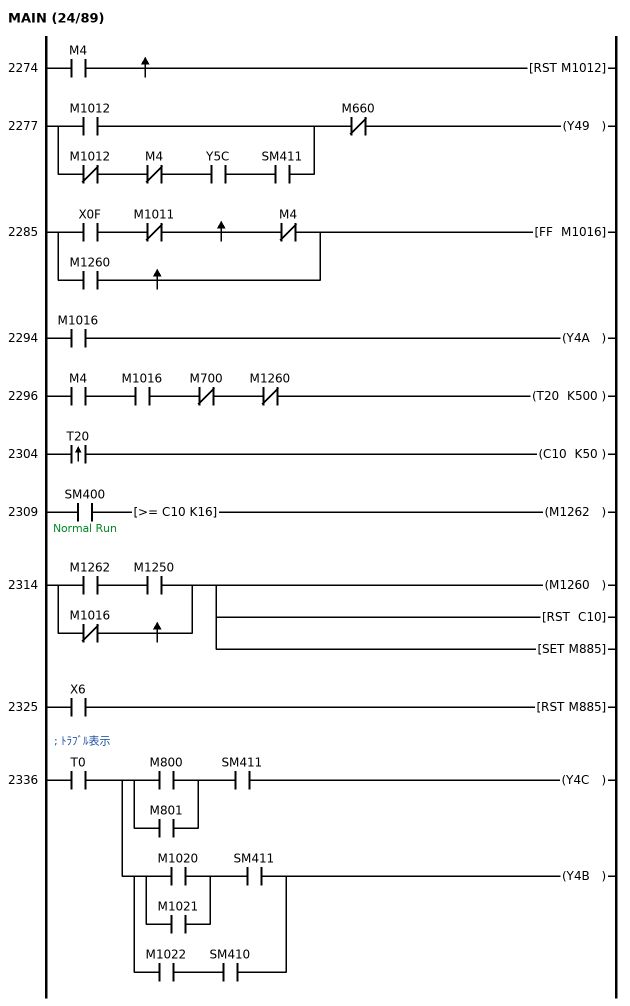
2274  LD      M4
      MEP
      RST     M1012
2277  LD      M1012
      LDI     M1012
      ANI     M4
      AND     Y5C
      AND     SM411
      ORB
      ANI     M660
      OUT     Y49
2285  LD      X0F
      ANI     M1011
      MEP
      ANI     M4
      LD      M1260
      MEP
      ORB
      FF      M1016
2294  LD      M1016
      OUT     Y4A
2296  LD      M4
      AND     M1016
      ANI     M700
      ANI     M1260
      OUT     T20 K500
2304  LDP     T20
      OUT     C10 K50
2309  LD      SM400  ; Normal Run
      AND>=   C10 K16
      OUT     M1262
2314  LD      M1262
      AND     M1250
      LDI     M1016
      MEP
      ORB
      OUT     M1260
      RST     C10
      SET     M885
2325  LD      X6
      RST     M885
; ﾄﾗﾌﾞﾙ表示
2336  LD      T0
      MPS
      LD      M800
      OR      M801
      ANB
      AND     SM411
      OUT     Y4C
      MPP
      LD      M1020
      OR      M1021
      AND     SM411
      LD      M1022
      AND     SM410
      ORB
      ANB
      OUT     Y4B
